KUKA KRL data list: 1234.dat

&ACCESS RVO
DEFDAT 1234
;FOLD EXTERNAL DECLARATIONS;%{PE}%MKUKATPBASIS,%CEXT,%VCOMMON,%P
  ;FOLD BASISTECH EXT;%{PE}%MKUKATPBASIS,%CEXT,%VEXT,%P
    EXT  BAS (BAS_COMMAND  :IN,REAL  :IN )
  ;ENDFOLD (BASISTECH EXT)

;ENDFOLD (EXTERNAL DECLARATIONS)
ENDDAT
